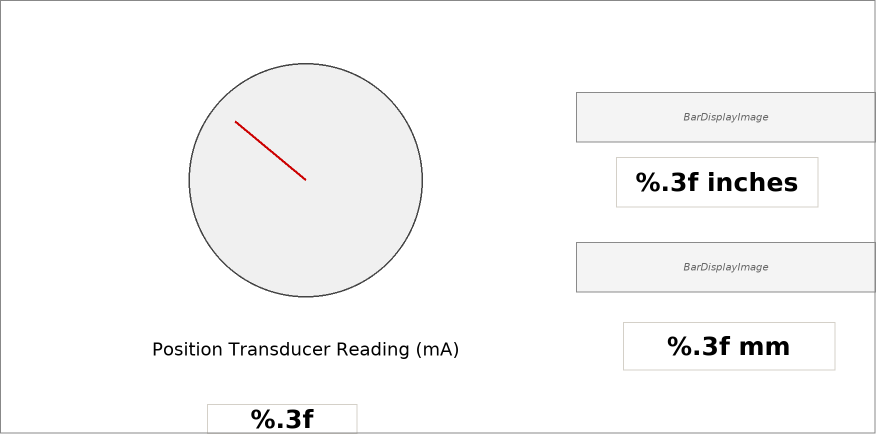
VISUALIZATION PositionTrans  // 876x434
    Meter360 (187,63 237x234), value: GVL.rCurrent_Input1_EU, style: Meter-Meter360-Gray, scale format: %.1f, scale 0..20
    Textfield (128,315 356x69), "Position Transducer Reading (mA)"
    Textfield (207,404 150x30), "%.3f", text variable: GVL.rCurrent_Input1_EU
    BarDisplayImage (576,92 300x50), style: BarDisplayImage-Gray, scale format: %.1f, scale 0..100
    BarDisplayImage (576,242 300x50), style: BarDisplayImage-Gray, scale format: %.1f, scale 0..100
    Textfield (616,157 202x50), "%.3f inches", text variable: MAIN.rPosSenDis_inch
    Textfield (623,322 212x48), "%.3f mm", text variable: MAIN.rPosSenDis_mm
END_VISUALIZATION

(* stored: Version 1.1.0.1, ProductVersion 3.1.4024.12
   Visu PositionTrans: Id {f4895278-4c84-4460-a50c-9e8ac8b23c1a} *)
